# EPICS autosave request: iocBoot/iocNSLS2_MIO/auto_settings.req
file "NSLS2_MIO_settings.req",          P=$(P), R=$(R)
file "quadEM_settings.req",            P=$(P), R=$(R)
file "quadEM_Plugin_settings.req",     P=$(P), R=$(R)
